FUNCTION alg_s_Dinitialized : BOOL
VAR_INPUT
	state: STATE;
END_VAR

alg_s_Dinitialized := (state.dvar_M_HardwareMap) = (elit_initialized);

END_FUNCTION

(* stored: Version 1.1.0.1, ProductVersion 3.1.4022.18
   POU alg_s_Dinitialized: Id {a98a079f-75fd-4ecc-85d5-14c390fe7292}, SpecialFunc None *)
